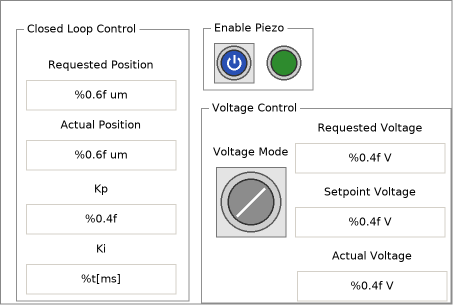
VISUALIZATION PiezoControls  // 453x305
VAR_IN_OUT
	Piezo	:	ST_PiezoAxis;
	ActPos	:	ST_HOMSStepper;
END_VAR
    GroupBox (203,20 110x70), "Enable Piezo"
        PowerSwitch (11,23 40x40), variable: Piezo.xEnable, behaviour: TOGGLE, style: Switch-PowerSwitch-Blue
        Lamp1 (61,23 40x40), variable: Piezo.xEnable and NOT Piezo.xError, style: Lamp-Lamp1-Green
    GroupBox (16,21 173x280), "Closed Loop Control"
        Textfield (10,59 150x30), "%0.6f um", text variable: Piezo.rReqAbsPos
            OnMouseClick: write the text variable via Default
        Textfield (10,119 150x30), "%0.6f um", text variable: ActPos.stAxis.NcToPlc.ActPos
        Label (10,89 150x30), "Actual Position"
        Label (10,29 150x30), "Requested Position"
        Textfield (10,183 150x30), "%0.4f", text variable: Piezo.stPIParams.fKp
            OnMouseClick: write the text variable via Default
        Textfield (10,243 150x30), "%t[ms]", text variable: Piezo.stPIParams.tTn
            OnMouseClick: write the text variable via Edit
        Label (10,153 150x30), "Kp"
        Label (10,213 150x30), "Ki"
    GroupBox (201,100 250x203), "Voltage Control"
        Textfield (94,43 150x30), "%0.4f V", text variable: Piezo.rReqVoltage
            OnMouseClick: write the text variable via Default
        Label (94,13 150x30), "Requested Voltage"
        Textfield (94,107 150x30), "%0.4f V", text variable: Piezo.rSetVoltage
        Label (94,77 150x30), "Setpoint Voltage"
        RotarySwitch (15,67 70x70), tooltip "Voltage mode", variable: Piezo.xVoltageMode, behaviour: TOGGLE, style: Switch-RotarySwitch-Gray
        Label (5,37 90x30), "Voltage Mode"
        Label (96,141 150x30), "Actual Voltage"
        Textfield (96,171 150x30), "%0.4f V", text variable: Piezo.rActVoltage
END_VISUALIZATION

(* stored: Version 1.1.0.1, ProductVersion 3.1.4020.12
   Visu PiezoControls: Id {6c39d4cc-2bd9-4c3a-9cf9-32254a64dc42} *)
